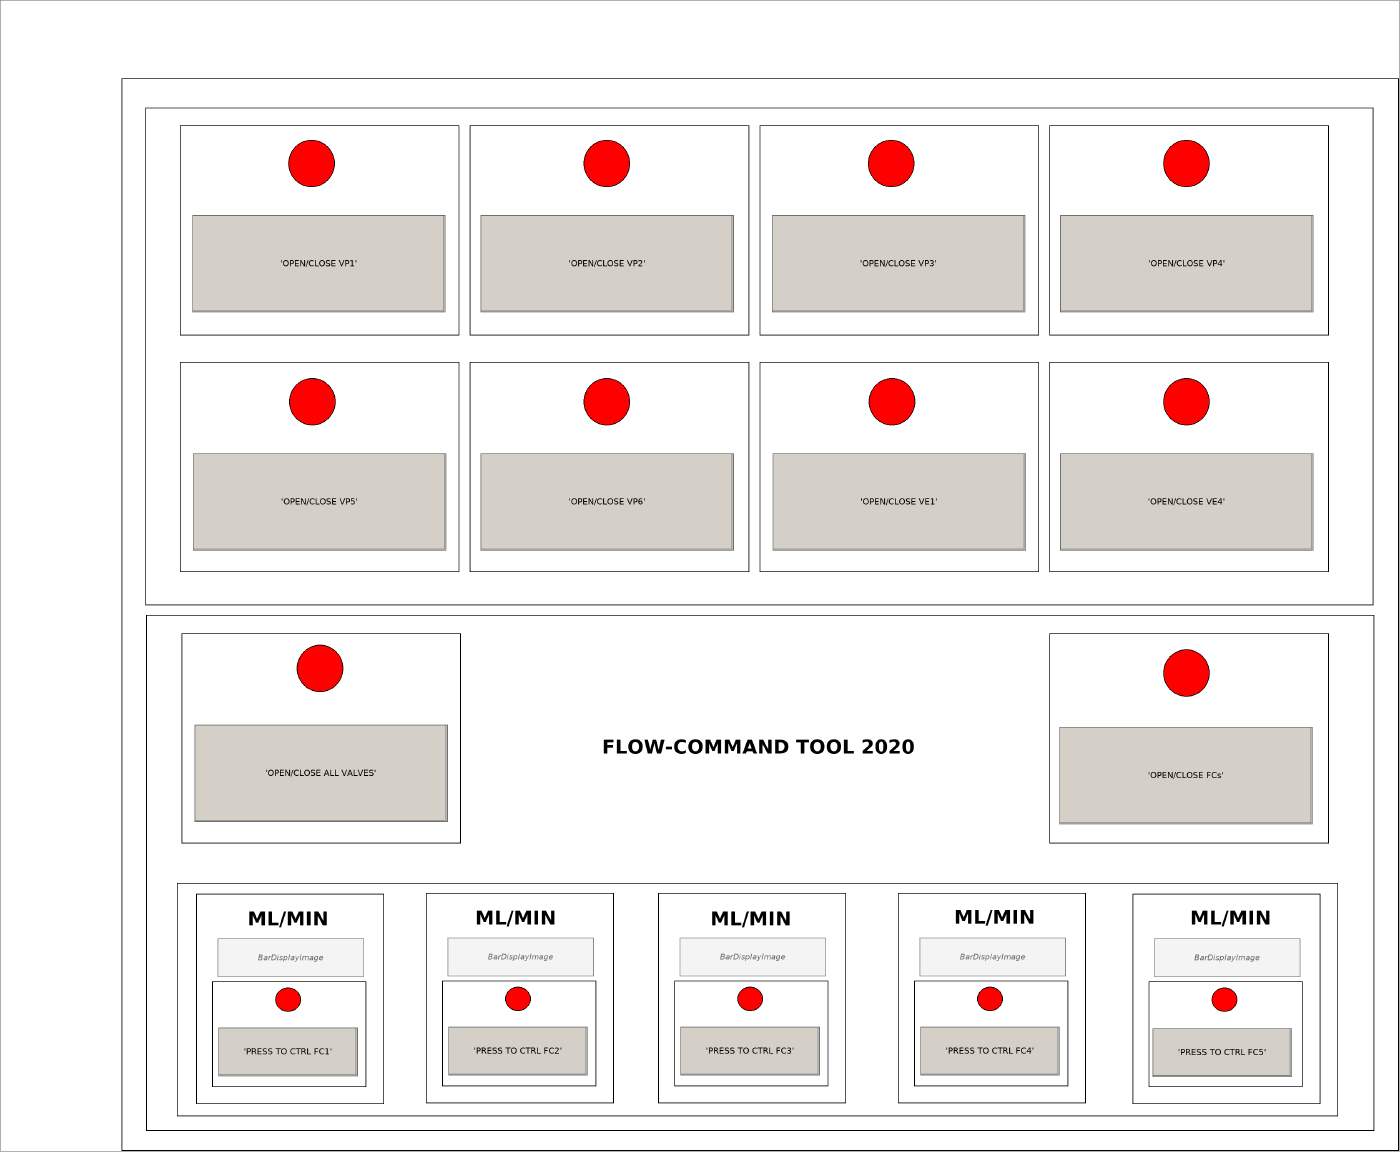
VISUALIZATION Visualization_1  // 1821x1499
    Rectangle (158,102 1661x1395)
    Rectangle (190,800 1597x671)
    Rectangle (230,1149 1510x303)
    Rectangle (189,140 1597x647)
    RoundedRectangle (611,471 363x273)
    RoundedRectangle (234,471 363x273)
    RoundedRectangle (611,163 363x273)
    RoundedRectangle (234,163 363x273)
    Ellipse (375,182 60x61), colour toggle: IO.r1_REF
    Button (250,280 329x126), "'OPEN/CLOSE VP1'"
        OnMouseClick: toggle IO.r1_REF
    Ellipse (759,182 60x61), colour toggle: IO.r2_REF
    Button (625,280 329x126), "'OPEN/CLOSE VP2'"
        OnMouseClick: toggle IO.r2_REF
    Ellipse (376,492 60x61), colour toggle: IO.r5_REF
    Button (251,590 329x126), "'OPEN/CLOSE VP5'"
        OnMouseClick: toggle IO.r5_REF
    Ellipse (759,492 60x61), colour toggle: IO.r6_REF
    Button (625,590 329x126), "'OPEN/CLOSE VP6'"
        OnMouseClick: toggle IO.r6_REF
    RoundedRectangle (255,1163 244x273)
    RoundedRectangle (276,1277 200x137)
    Button (284,1337 181x63), "'PRESS TO CTRL FC1'"
        OnMouseClick: toggle IO.p1_REF
    Ellipse (358,1285 33x31), colour toggle: IO.p1_REF
    BarDisplayImage (283,1221 190x50), value: MAIN.meter1, style: BarDisplayImage-Gray, scale format: %.1f, scale 0..500
    RoundedRectangle (1365,471 363x273)
    RoundedRectangle (988,471 363x273)
    RoundedRectangle (1365,163 363x273)
    RoundedRectangle (988,163 363x273)
    Ellipse (1129,182 60x61), colour toggle: IO.r3_REF
    Button (1004,280 329x126), "'OPEN/CLOSE VP3'"
        OnMouseClick: toggle IO.r3_REF
    Ellipse (1513,182 60x61), colour toggle: IO.r4_REF
    Button (1379,280 329x126), "'OPEN/CLOSE VP4'"
        OnMouseClick: toggle IO.r4_REF
    Ellipse (1130,492 60x61), colour toggle: IO.v1_REF
    Button (1005,590 329x126), "'OPEN/CLOSE VE1'"
        OnMouseClick: toggle IO.v1_REF
    Ellipse (1513,492 60x61), colour toggle: IO.v2_REF
    Button (1379,590 329x126), "'OPEN/CLOSE VE4'"
        OnMouseClick: toggle IO.v2_REF
    RoundedRectangle (236,824 363x273)
    Button (253,943 329x126), "'OPEN/CLOSE ALL VALVES'"
        OnMouseClick: toggle IO.erikoismuuttujaSum
    Ellipse (386,839 60x61), colour toggle: IO.erikoismuuttujaSum
    RoundedRectangle (1365,824 363x273)
    Ellipse (1513,845 60x61), colour toggle: IO.fx1_REF
    Button (1378,946 329x126), "'OPEN/CLOSE FCs'"
        OnMouseClick: toggle IO.fx1_REF
        OnMouseClick: toggle IO.fx2_REF
        OnMouseClick: toggle IO.fx3_REF
        OnMouseClick: toggle IO.fx4_REF
        OnMouseClick: toggle IO.fx5_REF
    RoundedRectangle (554,1162 244x273)
    RoundedRectangle (575,1276 200x137)
    Button (583,1336 181x63), "'PRESS TO CTRL FC2'"
        OnMouseClick: toggle IO.p2_REF
    Ellipse (657,1284 33x31), colour toggle: IO.p1_REF
    BarDisplayImage (582,1220 190x50), value: MAIN.meter2, style: BarDisplayImage-Gray, scale format: %.1f, scale 0..500
    RoundedRectangle (1473,1163 244x273)
    RoundedRectangle (1494,1277 200x137)
    Button (1499,1338 181x63), "'PRESS TO CTRL FC5'"
        OnMouseClick: toggle IO.p5_REF
    Ellipse (1576,1285 33x31), colour toggle: IO.p1_REF
    BarDisplayImage (1501,1221 190x50), value: MAIN.meter5, style: BarDisplayImage-Gray, scale format: %.1f, scale 0..500
    RoundedRectangle (1168,1162 244x273)
    RoundedRectangle (1189,1276 200x137)
    Button (1197,1336 181x63), "'PRESS TO CTRL FC4'"
        OnMouseClick: toggle IO.p4_REF
    Ellipse (1271,1284 33x31), colour toggle: IO.p1_REF
    BarDisplayImage (1196,1220 190x50), value: MAIN.meter4, style: BarDisplayImage-Gray, scale format: %.1f, scale 0..500
    RoundedRectangle (856,1162 244x273)
    RoundedRectangle (877,1276 200x137)
    Button (885,1336 181x63), "'PRESS TO CTRL FC3'"
        OnMouseClick: toggle IO.p3_REF
    Ellipse (959,1284 33x31), colour toggle: IO.p1_REF
    BarDisplayImage (884,1220 190x50), value: MAIN.meter3, style: BarDisplayImage-Gray, scale format: %.1f, scale 0..500
    Label (663,909 647x125), "FLOW-COMMAND TOOL 2020"
    Label (300,1180 150x30), "ML/MIN"
    Label (596,1179 150x30), "ML/MIN"
    Label (902,1180 150x30), "ML/MIN"
    Label (1219,1178 150x30), "ML/MIN"
    Label (1526,1179 150x30), "ML/MIN"
END_VISUALIZATION

(* stored: Version 1.1.0.1, ProductVersion 3.1.4024.0
   Visu Visualization_1: Id {92402780-3208-4360-9dcb-7b60ec972095} *)
